Fanuc KAREL source: ke00003.KL

-- PROVISIONAL review KL for V770-1; original PC SHA256 6ffd33b0ce8892f03fb58994a9586c8ec9dd547c5f9145fde61e7ce656577e77
-- Incomplete behavior may be omitted. Consult companion uncertainty JSON. Do not deploy.
PROGRAM KE00003
%NOLOCKGROUP
BEGIN
  -- UNRESOLVED_PC offsets 5-12; opcodes 9D,23
  -- UNRESOLVED_PC offsets 17-29; opcodes 3F,75
  -- UNRESOLVED_PC offsets 34-58; opcodes 27,22,22,2A,22,31
  -- UNRESOLVED_PC offsets 63-67; opcodes 7F
END KE00003
